// TIA Portal V17 export
Screen "Codex_Button_Test"  1280x740, Number=2
  ScreenLayer 
    Button "Codex_Button_1" at 100,100 size 220x80  Mode=Text, TextOff="Button", TextOn="Button"
